FUNCTION_BLOCK FB_UltraSonicSensor EXTENDS FB_NivelSensor
VAR_INPUT
END_VAR
VAR_OUTPUT
END_VAR
VAR

END_VAR

{warning 'Agregar implementación de método'}
METHOD Scale : BOOL
ScaledAnalog := AnalogSignal * MaxValue / 2000;
END_METHOD

END_FUNCTION_BLOCK

(* stored: Version 1.1.0.1, ProductVersion 3.1.4024.12
   POU FB_UltraSonicSensor: Id {f192cad1-2b8f-4ad8-a2d2-5b7934e29d7b}, SpecialFunc None
   Method Scale: Id {e54689f2-4b3e-41a7-9d98-911851e1da59} *)
